{attribute 'qualified_only' := ''}
{attribute 'strict' := ''}
TYPE cPuckStatusEval :
(
	None := 0
) DINT;
END_TYPE

(* stored: Version 1.1.0.1, ProductVersion 3.1.4024.6
   DUT cPuckStatusEval: Id {a452fbf6-2fff-42eb-9df0-1a2efffd72a2} *)
